TYPE BaseConfiguration :
STRUCT
	sName : STRING;
	sOutputDescription : STRING;
	sMountingPoint : STRING;
END_STRUCT
END_TYPE

(* stored: Version 1.1.0.1
   DUT BaseConfiguration: Id {b3d9baa8-9ada-47bf-a2f7-03853fd28a64} *)
